/// machine data that is used through most sequences of the unit (motor speed, axes positions, ...)
TYPE HandlingDataMachine :
STRUCT
  Slowspeed : LREAL;
  Highspeed : LREAL;
END_STRUCT
END_TYPE

(* stored: Version 1.1.0.1
   DUT HandlingDataMachine: Id {390e1e92-4523-40fd-b7f5-553632e8254a} *)
